// TIA Portal project "w1_button_led" (V14)

(* hardware
DEVICE "S7-1200 station_1"  S7-1200 Station
   slot 0: "Rack_0"  S7-1200 Rack  Rack  V1.0
   slot 1: "PLC_1"  CPU 1214C DC/DC/DC  6ES7 214-1AG40-0XB0  V4.2
*)

// ===== PLC "PLC_1"  CPU 1214C DC/DC/DC =====

VAR_GLOBAL   // PLC tag table "Default tag table"
   "D1" AT %Q0.0 : Bool;
   "D2" AT %Q0.1 : Bool;
   "D3" AT %Q0.2 : Bool;
   "PB0" AT %I0.0 : Bool;
   "PB1" AT %I0.1 : Bool;
   "PB2" AT %I0.2 : Bool;
   "PB3" AT %I0.3 : Bool;
   "PB4" AT %I0.4 : Bool;
END_VAR

ORGANIZATION_BLOCK "Main"   // OB1, LAD, ProgramCycle
TITLE = "Main Program Sweep (Cycle)"
{ S7_Optimized_Access := 'TRUE' }
VERSION : 0.1
   VAR_INPUT
      Initial_Call : Bool;   // Initial call of this OB
      Remanence : Bool;   // =True, if remanent data are available
   END_VAR
BEGIN

REGION Network 1
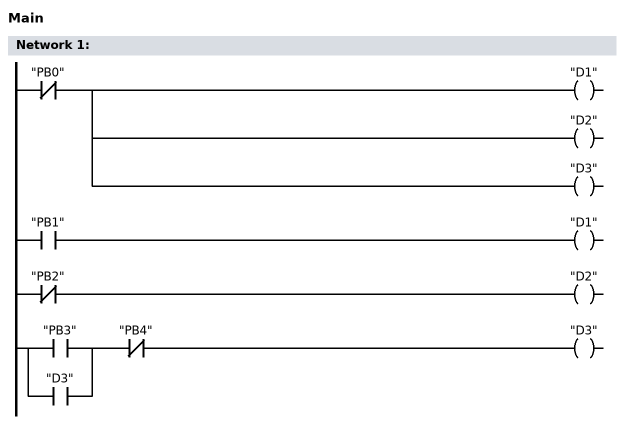
   RUNG wire#powerrail
      I_Contact( "PB0" )
      wire#w1
      Coil( "D1" )
   END_RUNG
   RUNG wire#w1
      Coil( "D2" )
   END_RUNG
   RUNG wire#w1
      Coil( "D3" )
   END_RUNG
   RUNG wire#powerrail
      Contact( "PB1" )
      Coil( "D1" )
   END_RUNG
   RUNG wire#powerrail
      I_Contact( "PB2" )
      Coil( "D2" )
   END_RUNG
   RUNG wire#powerrail
      Contact( "PB3" )
      wire#w2
      I_Contact( "PB4" )
      Coil( "D3" )
   END_RUNG
   RUNG wire#powerrail
      Contact( "D3" )
   END_RUNG wire#w2
   // the same network as SCL:
   "D1" := NOT "PB0";
   "D2" := NOT "PB0";
   "D3" := NOT "PB0";
   "D1" := "PB1";
   "D2" := NOT "PB2";
   "D3" := ("PB3" OR "D3") AND NOT "PB4";
END_REGION
END_ORGANIZATION_BLOCK